FUNCTION_BLOCK ABSTRACT Mc2MotionTask IMPLEMENTS I_Mc2MotionTask
VAR
	_Name : T_MaxString;
	_Axis : I_Mc2Axis;
END_VAR

PROPERTY Axis : I_Mc2Axis
GET
Axis := _Axis;
END_GET
SET
_Axis := Axis;
END_SET
END_PROPERTY

{attribute 'monitoring' := 'call'}
PROPERTY ABSTRACT Busy : BOOL
GET
END_GET
END_PROPERTY

METHOD ABSTRACT CyclicLogic
END_METHOD

{attribute 'monitoring' := 'call'}
PROPERTY ABSTRACT Error : BOOL
GET
END_GET
END_PROPERTY

{attribute 'monitoring' := 'call'}
PROPERTY ABSTRACT ErrorId : UDINT
GET
END_GET
END_PROPERTY

METHOD ABSTRACT Execute : BOOL;
END_METHOD

{attribute 'monitoring' := 'call'}
PROPERTY Name : T_MaxString
GET
Name := _Name;
END_GET
SET
_Name := Name;
END_SET
END_PROPERTY

END_FUNCTION_BLOCK

(* stored: Version 1.1.0.1, ProductVersion 3.1.4026.20
   POU Mc2MotionTask: Id {2a145b13-482c-4c39-9def-c2c0b08c225b}, SpecialFunc None
   Property Axis: Id {ed076f8d-b7d6-44f4-9870-51d18860c860}
   Get Get: Id {eb8068a9-6508-4c8c-9d7f-0d7599a8988b}
   Set Set: Id {42b420c4-9278-4267-80a1-964dc1f2d3de}
   Property Busy: Id {3d7b59fc-aef5-4abb-b38e-311755cfb5bc}
   Get Get: Id {5a89627e-65ac-4d75-9bbe-fb254369b00c}
   Method CyclicLogic: Id {9b3e73f8-b391-4bd9-ae12-fbe9eff82bd9}
   Property Error: Id {f4665e5f-790d-46ab-90f2-500638078a30}
   Get Get: Id {f8b6b48a-987b-4f59-9cd8-45fcdc31eb0b}
   Property ErrorId: Id {2e87e34c-91aa-4c8d-92e1-7c6b3905256f}
   Get Get: Id {b03956e9-6575-413f-b289-98035aef06b4}
   Method Execute: Id {1810cd75-364c-432d-b50a-2e9d60b60900}
   Property Name: Id {31afcebe-7038-4c40-8bf6-9c3f3ce58eea}
   Get Get: Id {0899c9d5-4249-46e5-b78b-6246087e897a}
   Set Set: Id {f923429b-7e41-4396-ba43-d116ddbbd378} *)
